TYPE E_MAA_States :
(
    Unknown := 0,
    Aprt1 := 1, //smallest
    Aprt2 := 2,
    Aprt3 := 3,
    Aprt4 := 4
);
END_TYPE

(* stored: Version 1.1.0.1, ProductVersion 3.1.4022.18
   DUT E_MAA_States: Id {9fa9f1d0-f1fd-4fbd-9ed0-3c2fdf5e1246} *)
